// TIA Portal V17 export
// export: Created 2023-12-22T15:05:34.8425877Z, ExportSetting WithDefaults, DisplayName Totally Integrated Automation Portal, DisplayVersion V17, DisplayName TIA Portal Openness, DisplayVersion V17, DisplayName TIA Portal Version Control Interface, DisplayVersion V17, DisplayName STEP 7 Professional, DisplayVersion V17, DisplayName STEP 7 Safety, DisplayVersion V17, DisplayName WinCC Advanced, DisplayVersion V17
DATA_BLOCK "Gaz_status_DB"   // DB3
VERSION : 0.1
// stored: AutoNumber true, DBAccessibleFromOPCUA true, InstanceOfName Gaz_status, InstanceOfType FB
"Gaz_status"
   // VAR
   //    Alarm : Word;
   //    H2_1_status : Int;
   //    H2_2_status : Int;
   //    Cl2_1_status : Int;
   //    Cl2_2_status : Int;
   // END_VAR
BEGIN
END_DATA_BLOCK
